Staubli VAL3: MENU.pgx

public program Menu(num x_nMenu, string x_sCustomTxt)
begin
  switch x_nMenu
    case 1
      cls()
      call BuildTitle(sListOfMessage[0],sOptionTitle)
      call up:type(0,1,"F1: 完整地校准(F2+F3)")
      call up:type(0,2,"F2: 校准编码器比例因数")
      call up:type(0,3,"F3: 校准传送带坐标系")
      call up:type(0,4,"F4: 校准视觉坐标系")
      //call up:type(0,5,"F5: Conveyor diagnostic")
      call up:type(0,6,"F6: 新建/加载传送带库")
      call up:type(0,7,"F7: 设置")
      call up:type(0,8,"F8: 结束")
      call up:type(10,10,"当前库: "+x_sCustomTxt)
      call up:typeMenu(1,"F1")
      call up:typeMenu(2,"F2")
      call up:typeMenu(3,"F3")
      call up:typeMenu(4,"F4")
      //call up:typeMenu(5, "F5")
      call up:typeMenu(6,"F6")
      call up:typeMenu(7,"F7")
      call up:typeMenu(8,"F8")
    break
    default
    break
  endSwitch
end
